// Mitsubishi GX Works2 project: R1R2 PLC Panel 20-08-2023_fr   PLC: Q03UDV

PROGRAM MAIN
; DEVICE NET
; OUTPUT LOGIC
; R1 TO R2 ZONE WAIT CLER
; R2 TO R1 ZONE
; CYCLE ON LOGIC
47    END
END_PROGRAM

PROGRAM CAMERA
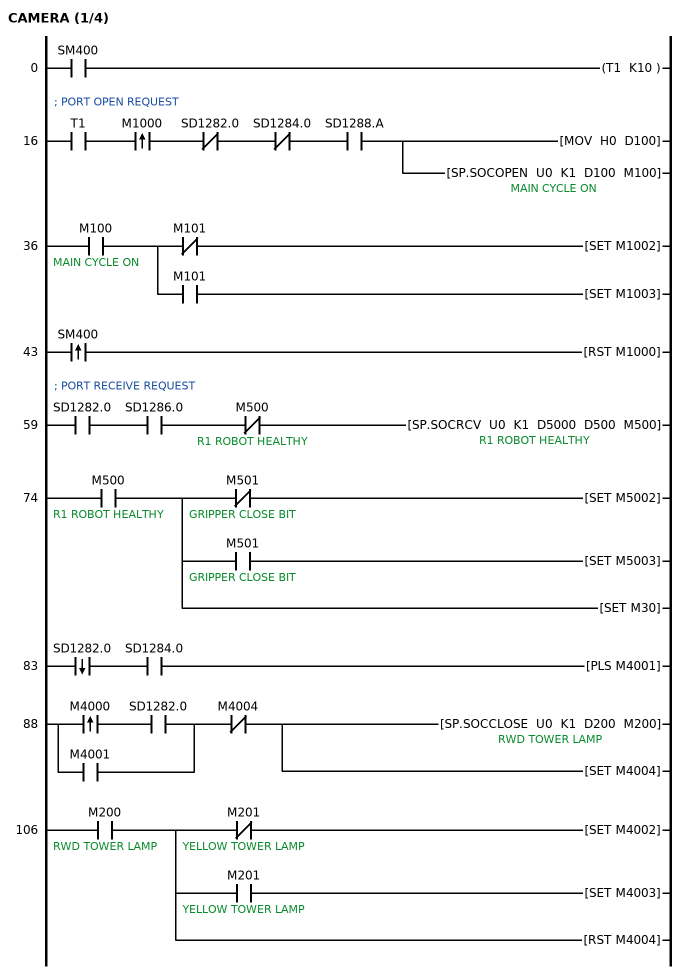
0     LD      SM400
      OUT     T1 K10
; PORT OPEN REQUEST
16    LD      T1
      ANDP    M1000
      ANI     SD1282.0
      ANI     SD1284.0
      AND     SD1288.A
      MOV     H0 D100
      SP.SOCOPEN U0 K1 D100 M100  ; MAIN CYCLE ON
36    LD      M100  ; MAIN CYCLE ON
      MPS
      ANI     M101
      SET     M1002
      MPP
      AND     M101
      SET     M1003
43    LDP     SM400
      RST     M1000
; PORT RECEIVE REQUEST
59    LD      SD1282.0
      AND     SD1286.0
      ANI     M500  ; R1 ROBOT HEALTHY
      SP.SOCRCV U0 K1 D5000 D500 M500
74    LD      M500  ; R1 ROBOT HEALTHY
      MPS
      ANI     M501  ; GRIPPER CLOSE BIT
      SET     M5002
      MRD
      AND     M501  ; GRIPPER CLOSE BIT
      SET     M5003
      MPP
      SET     M30
83    LDF     SD1282.0
      AND     SD1284.0
      PLS     M4001
88    LDP     M4000
      AND     SD1282.0
      OR      M4001
      ANI     M4004
      SP.SOCCLOSE U0 K1 D200 M200  ; RWD TOWER LAMP
      SET     M4004
106   LD      M200  ; RWD TOWER LAMP
      MPS
      ANI     M201  ; YELLOW TOWER LAMP
      SET     M4002
      MRD
      AND     M201  ; YELLOW TOWER LAMP
      SET     M4003
      MPP
      RST     M4004
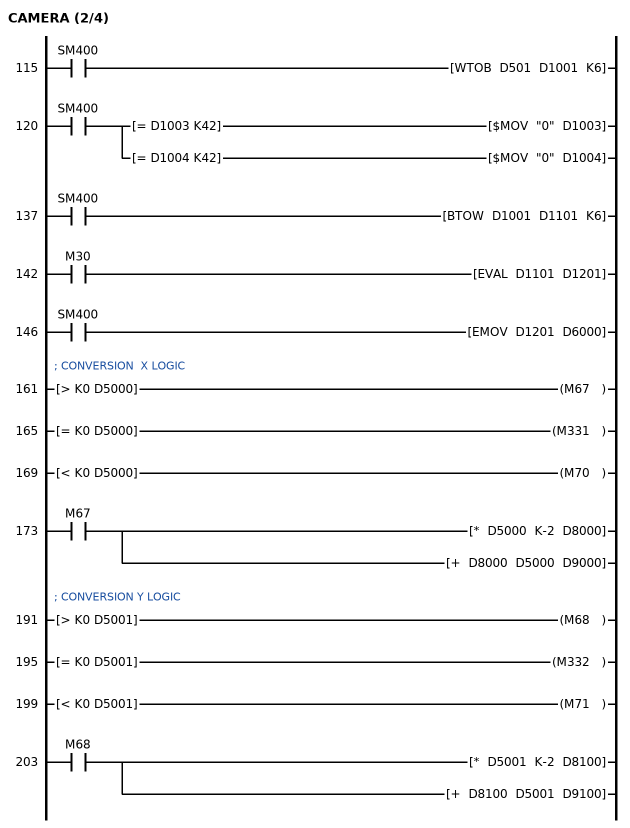
115   LD      SM400
      WTOB    D501 D1001 K6
120   LD      SM400
      MPS
      AND=    D1003 K42
      $MOV    "0" D1003
      MPP
      AND=    D1004 K42
      $MOV    "0" D1004
137   LD      SM400
      BTOW    D1001 D1101 K6
142   LD      M30
      EVAL    D1101 D1201
146   LD      SM400
      EMOV    D1201 D6000
; CONVERSION  X LOGIC
161   LD>     K0 D5000
      OUT     M67
165   LD=     K0 D5000
      OUT     M331
169   LD<     K0 D5000
      OUT     M70
173   LD      M67
      *       D5000 K-2 D8000
      +       D8000 D5000 D9000
; CONVERSION Y LOGIC
191   LD>     K0 D5001
      OUT     M68
195   LD=     K0 D5001
      OUT     M332
199   LD<     K0 D5001
      OUT     M71
203   LD      M68
      *       D5001 K-2 D8100
      +       D8100 D5001 D9100
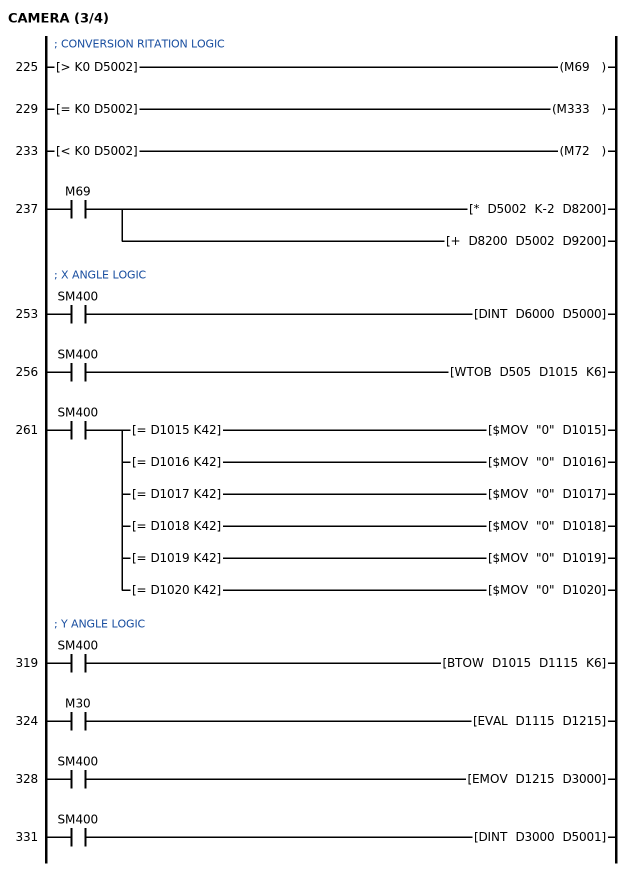
; CONVERSION RITATION LOGIC
225   LD>     K0 D5002
      OUT     M69
229   LD=     K0 D5002
      OUT     M333
233   LD<     K0 D5002
      OUT     M72
237   LD      M69
      *       D5002 K-2 D8200
      +       D8200 D5002 D9200
; X ANGLE LOGIC
253   LD      SM400
      DINT    D6000 D5000
256   LD      SM400
      WTOB    D505 D1015 K6
261   LD      SM400
      MPS
      AND=    D1015 K42
      $MOV    "0" D1015
      MRD
      AND=    D1016 K42
      $MOV    "0" D1016
      MRD
      AND=    D1017 K42
      $MOV    "0" D1017
      MRD
      AND=    D1018 K42
      $MOV    "0" D1018
      MRD
      AND=    D1019 K42
      $MOV    "0" D1019
      MPP
      AND=    D1020 K42
      $MOV    "0" D1020
; Y ANGLE LOGIC
319   LD      SM400
      BTOW    D1015 D1115 K6
324   LD      M30
      EVAL    D1115 D1215
328   LD      SM400
      EMOV    D1215 D3000
331   LD      SM400
      DINT    D3000 D5001
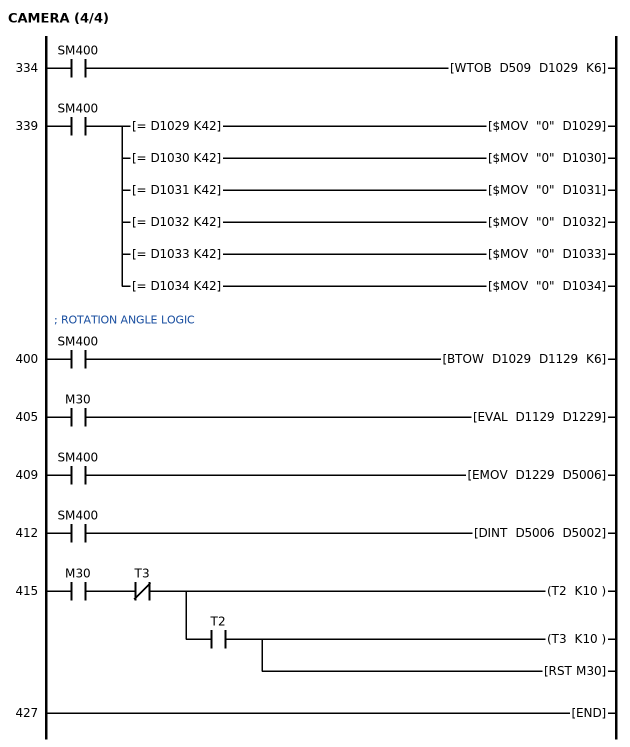
334   LD      SM400
      WTOB    D509 D1029 K6
339   LD      SM400
      MPS
      AND=    D1029 K42
      $MOV    "0" D1029
      MRD
      AND=    D1030 K42
      $MOV    "0" D1030
      MRD
      AND=    D1031 K42
      $MOV    "0" D1031
      MRD
      AND=    D1032 K42
      $MOV    "0" D1032
      MRD
      AND=    D1033 K42
      $MOV    "0" D1033
      MPP
      AND=    D1034 K42
      $MOV    "0" D1034
; ROTATION ANGLE LOGIC
400   LD      SM400
      BTOW    D1029 D1129 K6
405   LD      M30
      EVAL    D1129 D1229
409   LD      SM400
      EMOV    D1229 D5006
412   LD      SM400
      DINT    D5006 D5002
415   LD      M30
      ANI     T3
      OUT     T2 K10
      AND     T2
      OUT     T3 K10
      RST     M30
427   END
END_PROGRAM

PROGRAM AUTO
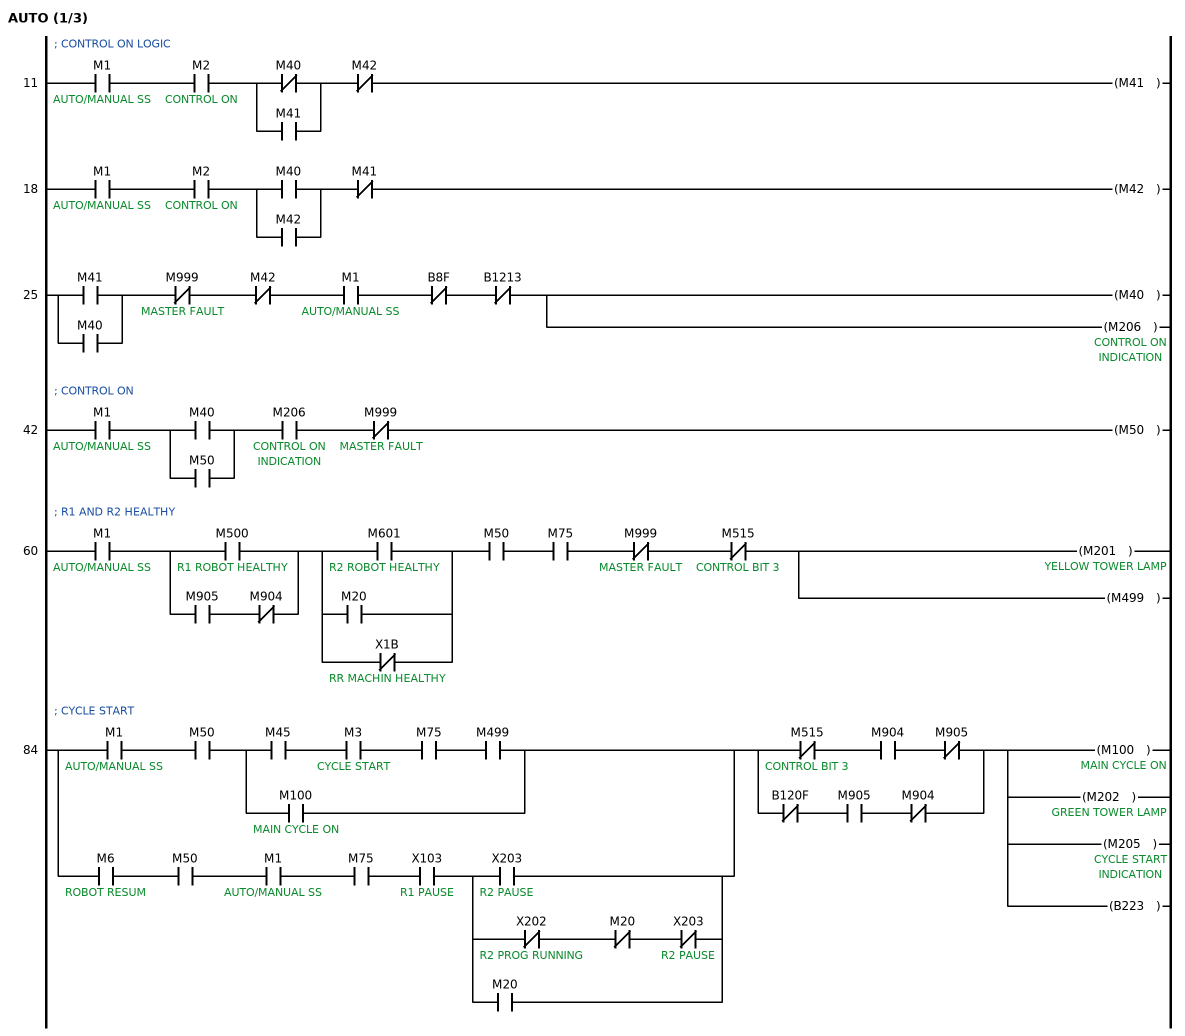
; CONTROL ON LOGIC
11    LD      M1  ; AUTO/MANUAL SS
      AND     M2  ; CONTROL ON
      LDI     M40
      OR      M41
      ANB
      ANI     M42
      OUT     M41
18    LD      M1  ; AUTO/MANUAL SS
      AND     M2  ; CONTROL ON
      LD      M40
      OR      M42
      ANB
      ANI     M41
      OUT     M42
25    LD      M41
      OR      M40
      ANI     M999  ; MASTER FAULT
      ANI     M42
      AND     M1  ; AUTO/MANUAL SS
      ANI     B8F
      ANI     B1213
      OUT     M40
      OUT     M206  ; CONTROL ON INDICATION
; CONTROL ON
42    LD      M1  ; AUTO/MANUAL SS
      LD      M40
      OR      M50
      ANB
      AND     M206  ; CONTROL ON INDICATION
      ANI     M999  ; MASTER FAULT
      OUT     M50
; R1 AND R2 HEALTHY
60    LD      M1  ; AUTO/MANUAL SS
      LD      M500  ; R1 ROBOT HEALTHY
      LD      M905
      ANI     M904
      ORB
      ANB
      LD      M601  ; R2 ROBOT HEALTHY
      OR      M20
      ORI     X1B  ; RR MACHIN HEALTHY
      ANB
      AND     M50
      AND     M75
      ANI     M999  ; MASTER FAULT
      ANI     M515  ; CONTROL BIT 3
      OUT     M201  ; YELLOW TOWER LAMP
      OUT     M499
; CYCLE START
84    LD      M1  ; AUTO/MANUAL SS
      AND     M50
      LD      M45
      AND     M3  ; CYCLE START
      AND     M75
      AND     M499
      OR      M100  ; MAIN CYCLE ON
      ANB
      LD      M6  ; ROBOT RESUM
      AND     M50
      AND     M1  ; AUTO/MANUAL SS
      AND     M75
      AND     X103  ; R1 PAUSE
      LD      X203  ; R2 PAUSE
      LDI     X202  ; R2 PROG RUNNING
      ANI     M20
      ANI     X203  ; R2 PAUSE
      ORB
      OR      M20
      ANB
      ORB
      LDI     M515  ; CONTROL BIT 3
      AND     M904
      ANI     M905
      LDI     B120F
      AND     M905
      ANI     M904
      ORB
      ANB
      OUT     M100  ; MAIN CYCLE ON
      OUT     M202  ; GREEN TOWER LAMP
      OUT     M205  ; CYCLE START INDICATION
      OUT     B223
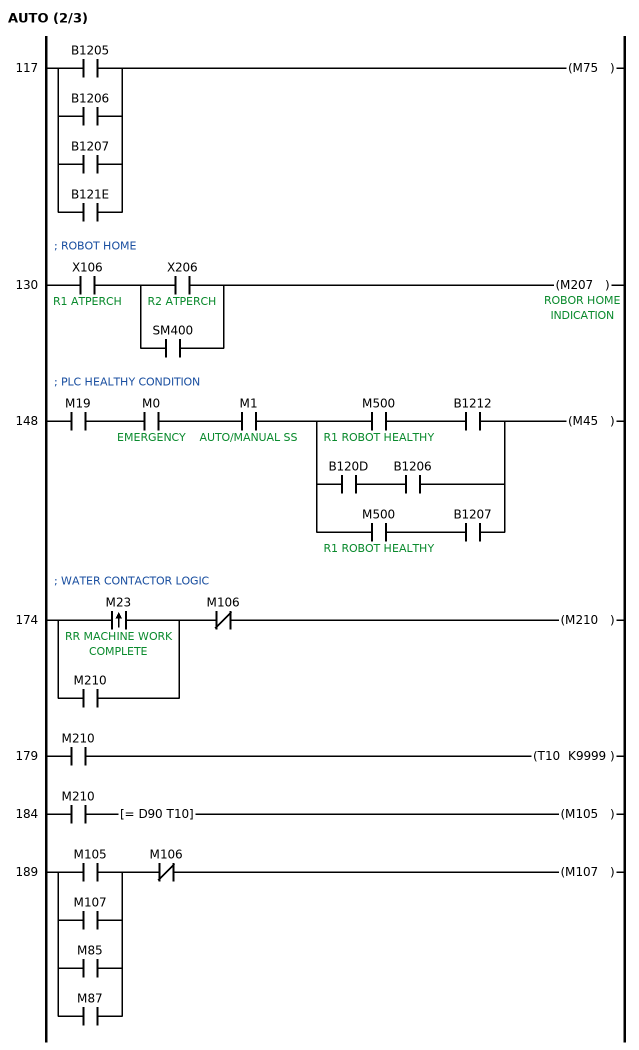
117   LD      B1205
      OR      B1206
      OR      B1207
      OR      B121E
      OUT     M75
; ROBOT HOME
130   LD      X106  ; R1 ATPERCH
      LD      X206  ; R2 ATPERCH
      OR      SM400
      ANB
      OUT     M207  ; ROBOR HOME INDICATION
; PLC HEALTHY CONDITION
148   LD      M19
      AND     M0  ; EMERGENCY
      AND     M1  ; AUTO/MANUAL SS
      LD      M500  ; R1 ROBOT HEALTHY
      AND     B1212
      LD      B120D
      AND     B1206
      ORB
      LD      M500  ; R1 ROBOT HEALTHY
      AND     B1207
      ORB
      ANB
      OUT     M45
; WATER CONTACTOR LOGIC
174   LDP     M23  ; RR MACHINE WORK COMPLETE
      OR      M210
      ANI     M106
      OUT     M210
179   LD      M210
      OUT     T10 K9999
184   LD      M210
      AND=    D90 T10
      OUT     M105
189   LD      M105
      OR      M107
      OR      M85
      OR      M87
      ANI     M106
      OUT     M107
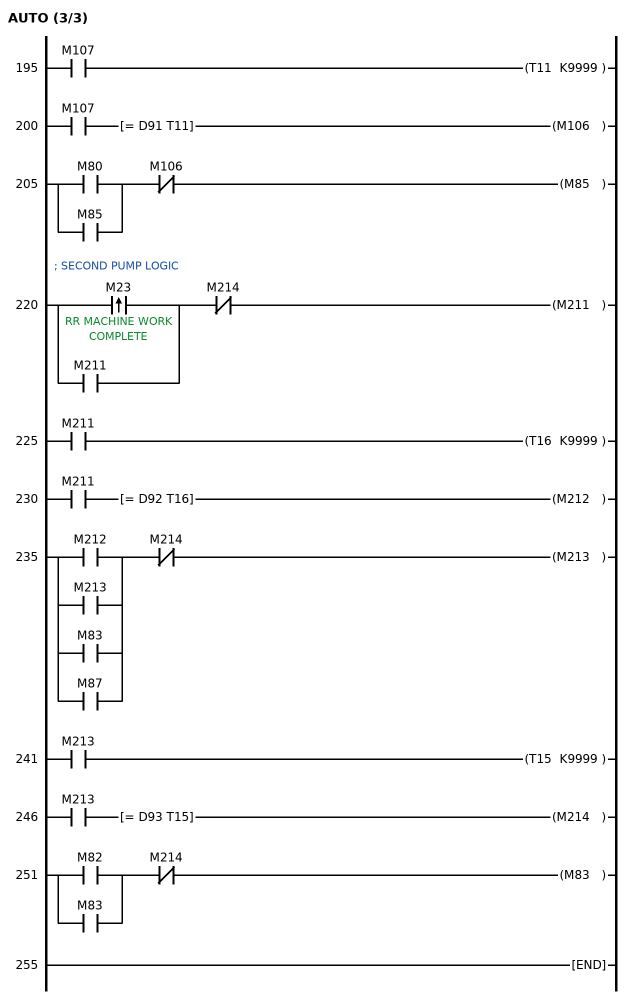
195   LD      M107
      OUT     T11 K9999
200   LD      M107
      AND=    D91 T11
      OUT     M106
205   LD      M80
      OR      M85
      ANI     M106
      OUT     M85
; SECOND PUMP LOGIC
220   LDP     M23  ; RR MACHINE WORK COMPLETE
      OR      M211
      ANI     M214
      OUT     M211
225   LD      M211
      OUT     T16 K9999
230   LD      M211
      AND=    D92 T16
      OUT     M212
235   LD      M212
      OR      M213
      OR      M83
      OR      M87
      ANI     M214
      OUT     M213
241   LD      M213
      OUT     T15 K9999
246   LD      M213
      AND=    D93 T15
      OUT     M214
251   LD      M82
      OR      M83
      ANI     M214
      OUT     M83
255   END
END_PROGRAM

PROGRAM CCLINK
0     END
END_PROGRAM

PROGRAM D-NET
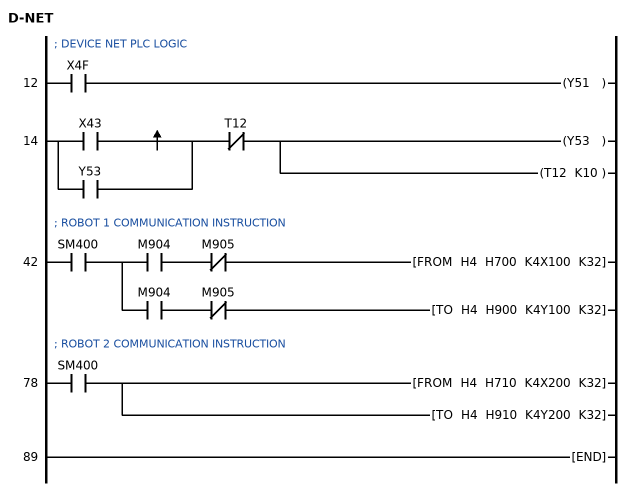
; DEVICE NET PLC LOGIC
12    LD      X4F
      OUT     Y51
14    LD      X43
      MEP
      OR      Y53
      ANI     T12
      OUT     Y53
      OUT     T12 K10
; ROBOT 1 COMMUNICATION INSTRUCTION
42    LD      SM400
      MPS
      AND     M904
      ANI     M905
      FROM    H4 H700 K4X100 K32  ; R1 CMD ENABLE
      MPP
      AND     M904
      ANI     M905
      TO      H4 H900 K4Y100 K32  ; R1 IMSTP
; ROBOT 2 COMMUNICATION INSTRUCTION
78    LD      SM400
      FROM    H4 H710 K4X200 K32  ; R2 CMD ENABLE
      TO      H4 H910 K4Y200 K32  ; R2 IMSTP
89    END
END_PROGRAM

PROGRAM FAULT
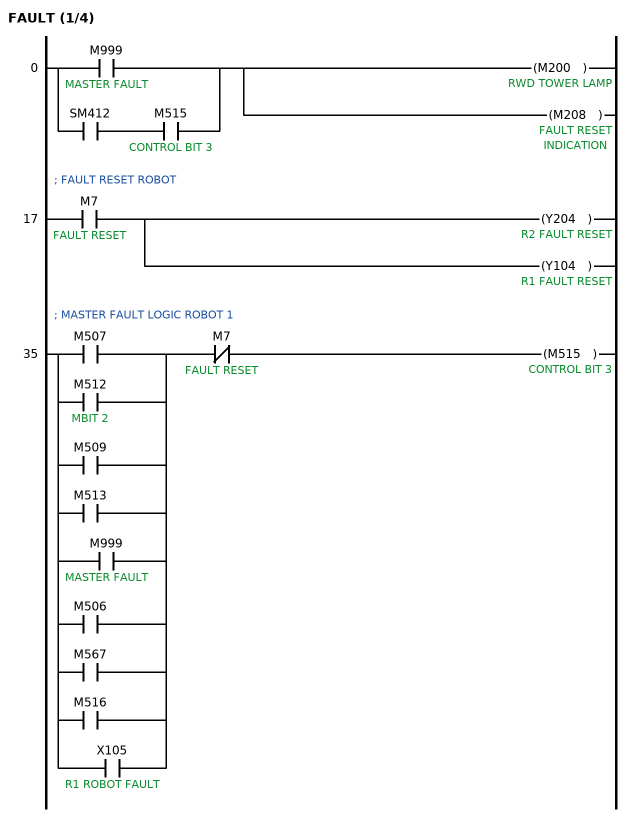
0     LD      M999  ; MASTER FAULT
      LD      SM412
      AND     M515  ; CONTROL BIT 3
      ORB
      OUT     M200  ; RWD TOWER LAMP
      OUT     M208  ; FAULT RESET INDICATION
; FAULT RESET ROBOT
17    LD      M7  ; FAULT RESET
      OUT     Y204  ; R2 FAULT RESET
      OUT     Y104  ; R1 FAULT RESET
; MASTER FAULT LOGIC ROBOT 1
35    LD      M507
      OR      M512  ; MBIT 2
      OR      M509
      OR      M513
      OR      M999  ; MASTER FAULT
      OR      M506
      OR      M567
      OR      M516
      OR      X105  ; R1 ROBOT FAULT
      ANI     M7  ; FAULT RESET
      OUT     M515  ; CONTROL BIT 3
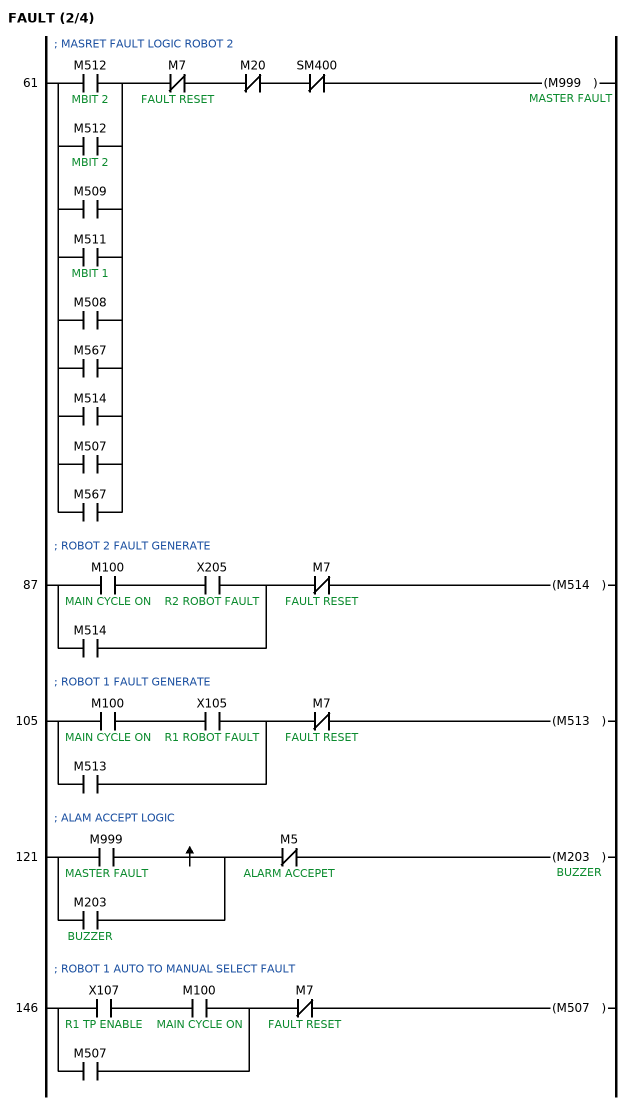
; MASRET FAULT LOGIC ROBOT 2
61    LD      M512  ; MBIT 2
      OR      M512  ; MBIT 2
      OR      M509
      OR      M511  ; MBIT 1
      OR      M508
      OR      M567
      OR      M514
      OR      M507
      OR      M567
      ANI     M7  ; FAULT RESET
      ANI     M20
      ANI     SM400
      OUT     M999  ; MASTER FAULT
; ROBOT 2 FAULT GENERATE
87    LD      M100  ; MAIN CYCLE ON
      AND     X205  ; R2 ROBOT FAULT
      OR      M514
      ANI     M7  ; FAULT RESET
      OUT     M514
; ROBOT 1 FAULT GENERATE
105   LD      M100  ; MAIN CYCLE ON
      AND     X105  ; R1 ROBOT FAULT
      OR      M513
      ANI     M7  ; FAULT RESET
      OUT     M513
; ALAM ACCEPT LOGIC
121   LD      M999  ; MASTER FAULT
      MEP
      OR      M203  ; BUZZER
      ANI     M5  ; ALARM ACCEPET
      OUT     M203  ; BUZZER
; ROBOT 1 AUTO TO MANUAL SELECT FAULT
146   LD      X107  ; R1 TP ENABLE
      AND     M100  ; MAIN CYCLE ON
      OR      M507
      ANI     M7  ; FAULT RESET
      OUT     M507
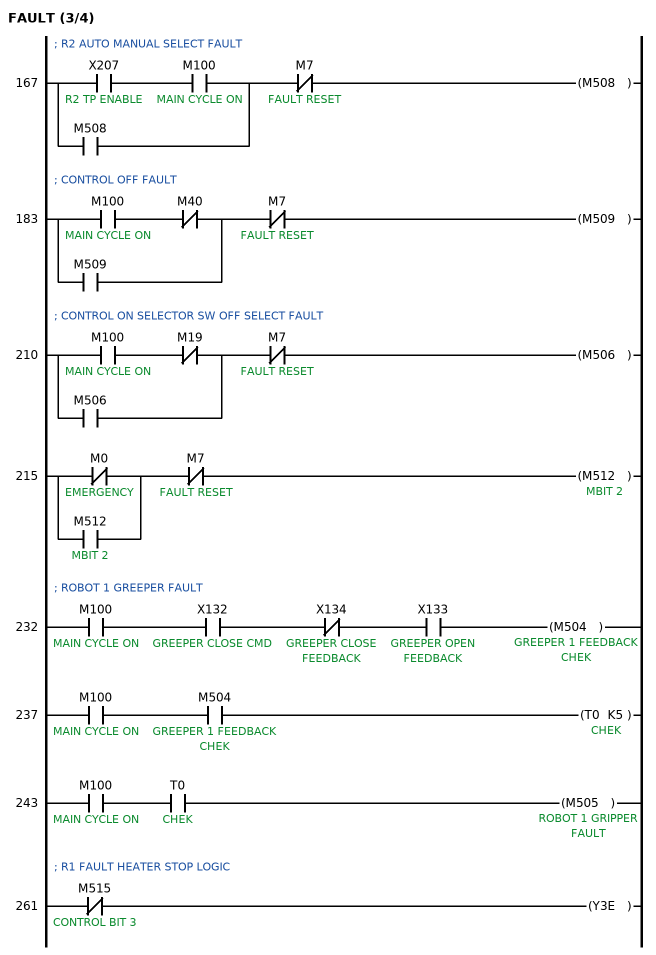
; R2 AUTO MANUAL SELECT FAULT
167   LD      X207  ; R2 TP ENABLE
      AND     M100  ; MAIN CYCLE ON
      OR      M508
      ANI     M7  ; FAULT RESET
      OUT     M508
; CONTROL OFF FAULT
183   LD      M100  ; MAIN CYCLE ON
      ANI     M40
      OR      M509
      ANI     M7  ; FAULT RESET
      OUT     M509
; CONTROL ON SELECTOR SW OFF SELECT FAULT
210   LD      M100  ; MAIN CYCLE ON
      ANI     M19
      OR      M506
      ANI     M7  ; FAULT RESET
      OUT     M506
215   LDI     M0  ; EMERGENCY
      OR      M512  ; MBIT 2
      ANI     M7  ; FAULT RESET
      OUT     M512  ; MBIT 2
; ROBOT 1 GREEPER FAULT
232   LD      M100  ; MAIN CYCLE ON
      AND     X132  ; GREEPER CLOSE CMD
      ANI     X134  ; GREEPER CLOSE FEEDBACK
      AND     X133  ; GREEPER OPEN FEEDBACK
      OUT     M504  ; GREEPER 1 FEEDBACK CHEK
237   LD      M100  ; MAIN CYCLE ON
      AND     M504  ; GREEPER 1 FEEDBACK CHEK
      OUT     T0 K5  ; CHEK
243   LD      M100  ; MAIN CYCLE ON
      AND     T0  ; CHEK
      OUT     M505  ; ROBOT 1 GRIPPER FAULT
; R1 FAULT HEATER STOP LOGIC
261   LDI     M515  ; CONTROL BIT 3
      OUT     Y3E
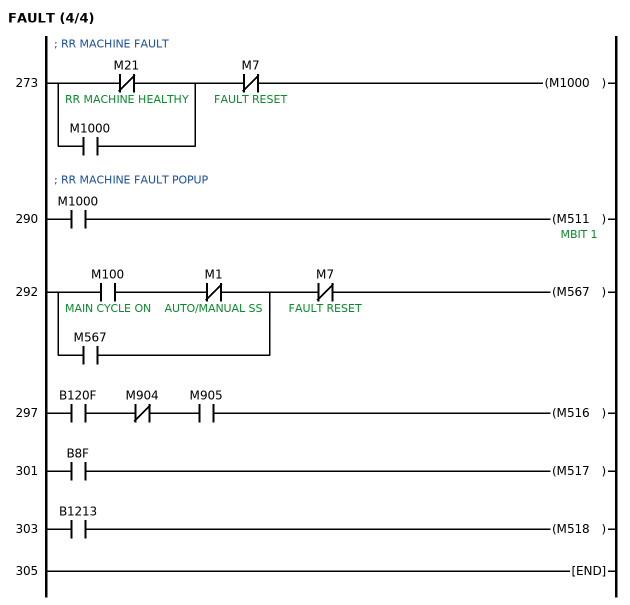
; RR MACHINE FAULT
273   LDI     M21  ; RR MACHINE HEALTHY
      OR      M1000
      ANI     M7  ; FAULT RESET
      OUT     M1000
; RR MACHINE FAULT POPUP
290   LD      M1000
      OUT     M511  ; MBIT 1
292   LD      M100  ; MAIN CYCLE ON
      ANI     M1  ; AUTO/MANUAL SS
      OR      M567
      ANI     M7  ; FAULT RESET
      OUT     M567
297   LD      B120F
      ANI     M904
      AND     M905
      OUT     M516
301   LD      B8F
      OUT     M517
303   LD      B1213
      OUT     M518
305   END
END_PROGRAM

PROGRAM INPUTMAP
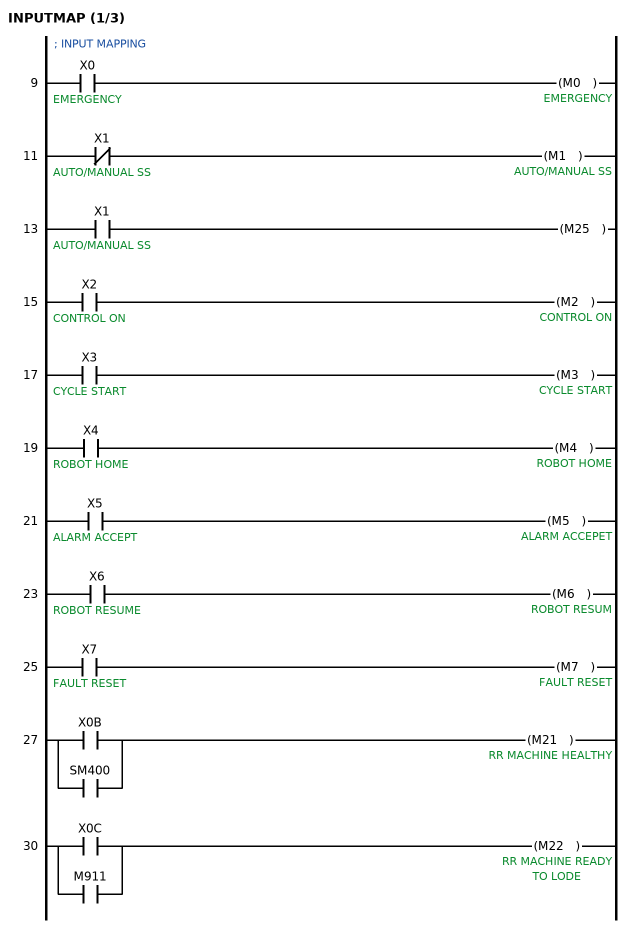
; INPUT MAPPING
9     LD      X0  ; EMERGENCY
      OUT     M0  ; EMERGENCY
11    LDI     X1  ; AUTO/MANUAL SS
      OUT     M1  ; AUTO/MANUAL SS
13    LD      X1  ; AUTO/MANUAL SS
      OUT     M25
15    LD      X2  ; CONTROL ON
      OUT     M2  ; CONTROL ON
17    LD      X3  ; CYCLE START
      OUT     M3  ; CYCLE START
19    LD      X4  ; ROBOT HOME
      OUT     M4  ; ROBOT HOME
21    LD      X5  ; ALARM ACCEPT
      OUT     M5  ; ALARM ACCEPET
23    LD      X6  ; ROBOT RESUME
      OUT     M6  ; ROBOT RESUM
25    LD      X7  ; FAULT RESET
      OUT     M7  ; FAULT RESET
27    LD      X0B
      OR      SM400
      OUT     M21  ; RR MACHINE HEALTHY
30    LD      X0C
      OR      M911
      OUT     M22  ; RR MACHINE READY TO LODE
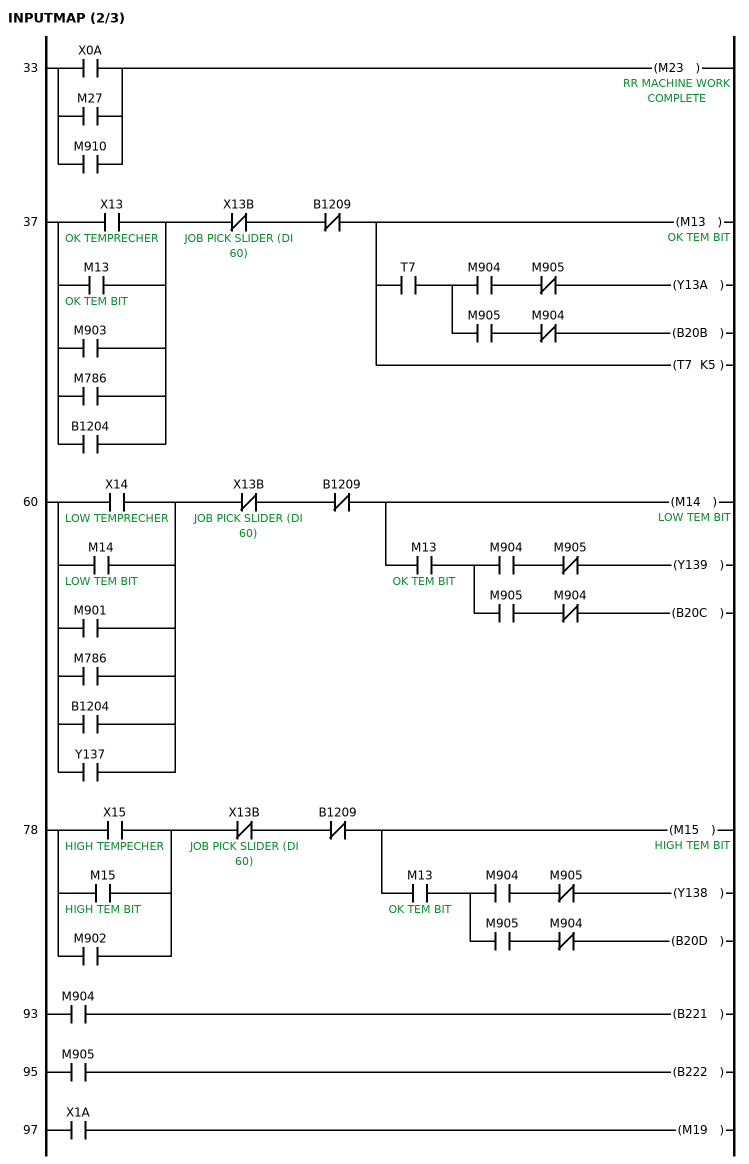
33    LD      X0A
      OR      M27
      OR      M910
      OUT     M23  ; RR MACHINE WORK COMPLETE
37    LD      X13  ; OK TEMPRECHER
      OR      M13  ; OK TEM BIT
      OR      M903
      OR      M786
      OR      B1204
      ANI     X13B  ; JOB PICK SLIDER (DI 60)
      ANI     B1209
      OUT     M13  ; OK TEM BIT
      MPS
      AND     T7
      MPS
      AND     M904
      ANI     M905
      OUT     Y13A
      MPP
      AND     M905
      ANI     M904
      OUT     B20B
      MPP
      OUT     T7 K5
60    LD      X14  ; LOW TEMPRECHER
      OR      M14  ; LOW TEM BIT
      OR      M901
      OR      M786
      OR      B1204
      OR      Y137
      ANI     X13B  ; JOB PICK SLIDER (DI 60)
      ANI     B1209
      OUT     M14  ; LOW TEM BIT
      AND     M13  ; OK TEM BIT
      MPS
      AND     M904
      ANI     M905
      OUT     Y139
      MPP
      AND     M905
      ANI     M904
      OUT     B20C
78    LD      X15  ; HIGH TEMPECHER
      OR      M15  ; HIGH TEM BIT
      OR      M902
      ANI     X13B  ; JOB PICK SLIDER (DI 60)
      ANI     B1209
      OUT     M15  ; HIGH TEM BIT
      AND     M13  ; OK TEM BIT
      MPS
      AND     M904
      ANI     M905
      OUT     Y138
      MPP
      AND     M905
      ANI     M904
      OUT     B20D
93    LD      M904
      OUT     B221
95    LD      M905
      OUT     B222
97    LD      X1A
      OUT     M19
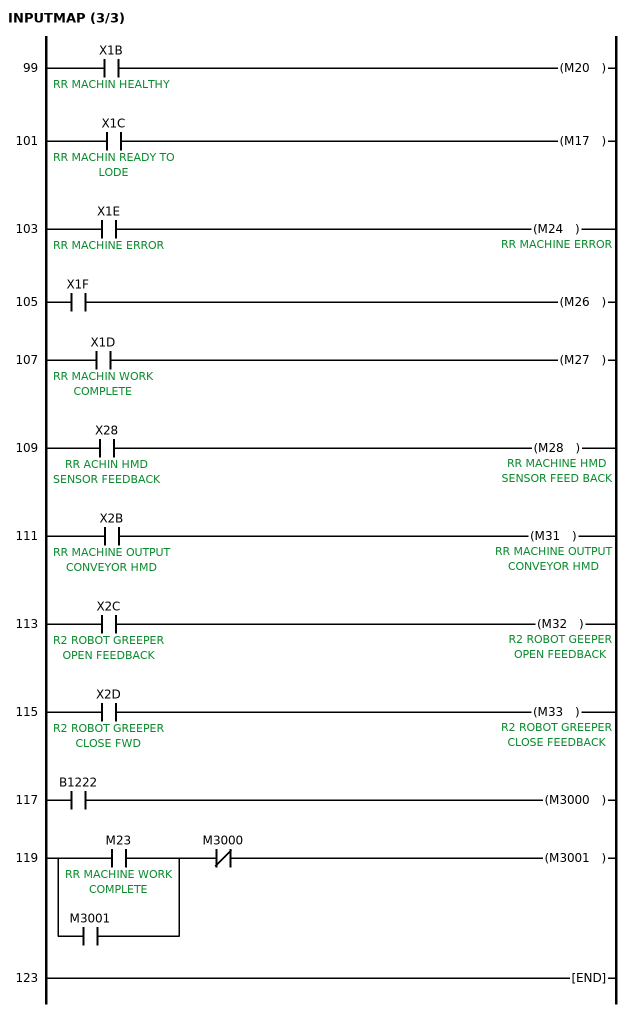
99    LD      X1B  ; RR MACHIN HEALTHY
      OUT     M20
101   LD      X1C  ; RR MACHIN READY TO LODE
      OUT     M17
103   LD      X1E  ; RR MACHINE ERROR
      OUT     M24  ; RR MACHINE ERROR
105   LD      X1F
      OUT     M26
107   LD      X1D  ; RR MACHIN WORK COMPLETE
      OUT     M27
109   LD      X28  ; RR ACHIN HMD SENSOR FEEDBACK
      OUT     M28  ; RR MACHINE HMD SENSOR FEED BACK
111   LD      X2B  ; RR MACHINE OUTPUT CONVEYOR HMD
      OUT     M31  ; RR MACHINE OUTPUT CONVEYOR HMD
113   LD      X2C  ; R2 ROBOT GREEPER OPEN FEEDBACK
      OUT     M32  ; R2 ROBOT GEEPER OPEN FEEDBACK
115   LD      X2D  ; R2 ROBOT GREEPER CLOSE FWD
      OUT     M33  ; R2 ROBOT GREEPER CLOSE FEEDBACK
117   LD      B1222
      OUT     M3000
119   LD      M23  ; RR MACHINE WORK COMPLETE
      OR      M3001
      ANI     M3000
      OUT     M3001
123   END
END_PROGRAM

PROGRAM MANUAL
0     END
END_PROGRAM

PROGRAM OUTPUTMA
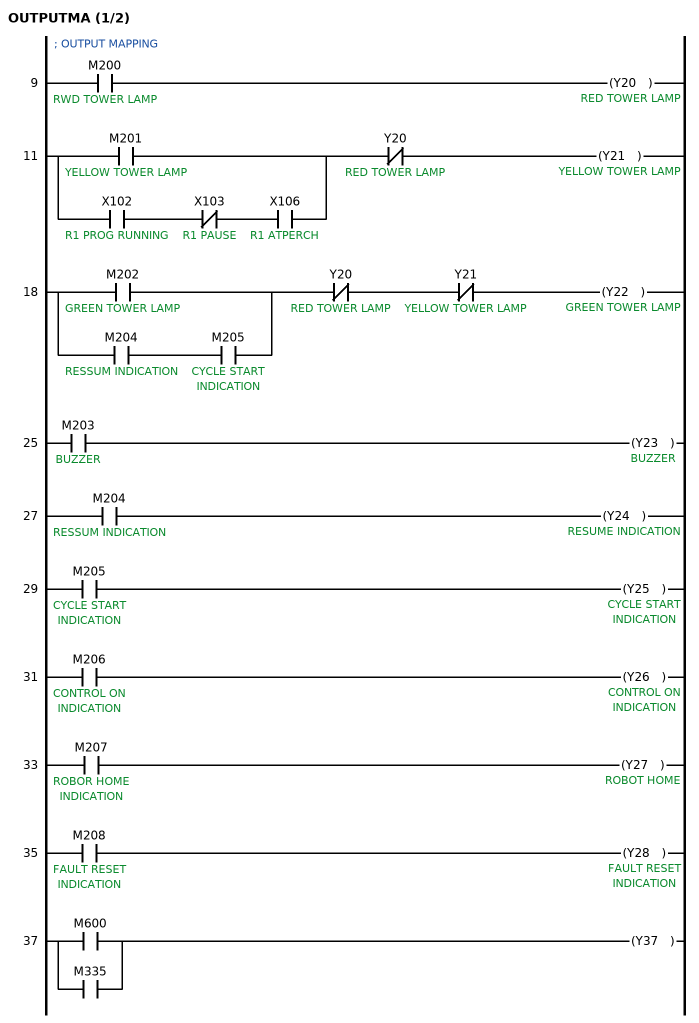
; OUTPUT MAPPING
9     LD      M200  ; RWD TOWER LAMP
      OUT     Y20  ; RED TOWER LAMP
11    LD      M201  ; YELLOW TOWER LAMP
      LD      X102  ; R1 PROG RUNNING
      ANI     X103  ; R1 PAUSE
      AND     X106  ; R1 ATPERCH
      ORB
      ANI     Y20  ; RED TOWER LAMP
      OUT     Y21  ; YELLOW TOWER LAMP
18    LD      M202  ; GREEN TOWER LAMP
      LD      M204  ; RESSUM INDICATION
      AND     M205  ; CYCLE START INDICATION
      ORB
      ANI     Y20  ; RED TOWER LAMP
      ANI     Y21  ; YELLOW TOWER LAMP
      OUT     Y22  ; GREEN TOWER LAMP
25    LD      M203  ; BUZZER
      OUT     Y23  ; BUZZER
27    LD      M204  ; RESSUM INDICATION
      OUT     Y24  ; RESUME INDICATION
29    LD      M205  ; CYCLE START INDICATION
      OUT     Y25  ; CYCLE START  INDICATION
31    LD      M206  ; CONTROL ON INDICATION
      OUT     Y26  ; CONTROL ON INDICATION
33    LD      M207  ; ROBOR HOME INDICATION
      OUT     Y27  ; ROBOT HOME
35    LD      M208  ; FAULT RESET INDICATION
      OUT     Y28  ; FAULT RESET INDICATION
37    LD      M600
      OR      M335
      OUT     Y37
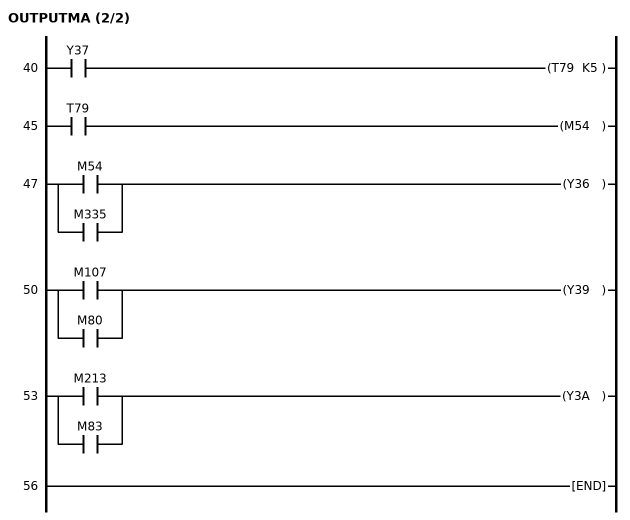
40    LD      Y37
      OUT     T79 K5
45    LD      T79
      OUT     M54
47    LD      M54
      OR      M335
      OUT     Y36
50    LD      M107
      OR      M80
      OUT     Y39
53    LD      M213
      OR      M83
      OUT     Y3A
56    END
END_PROGRAM

PROGRAM ROBO_1
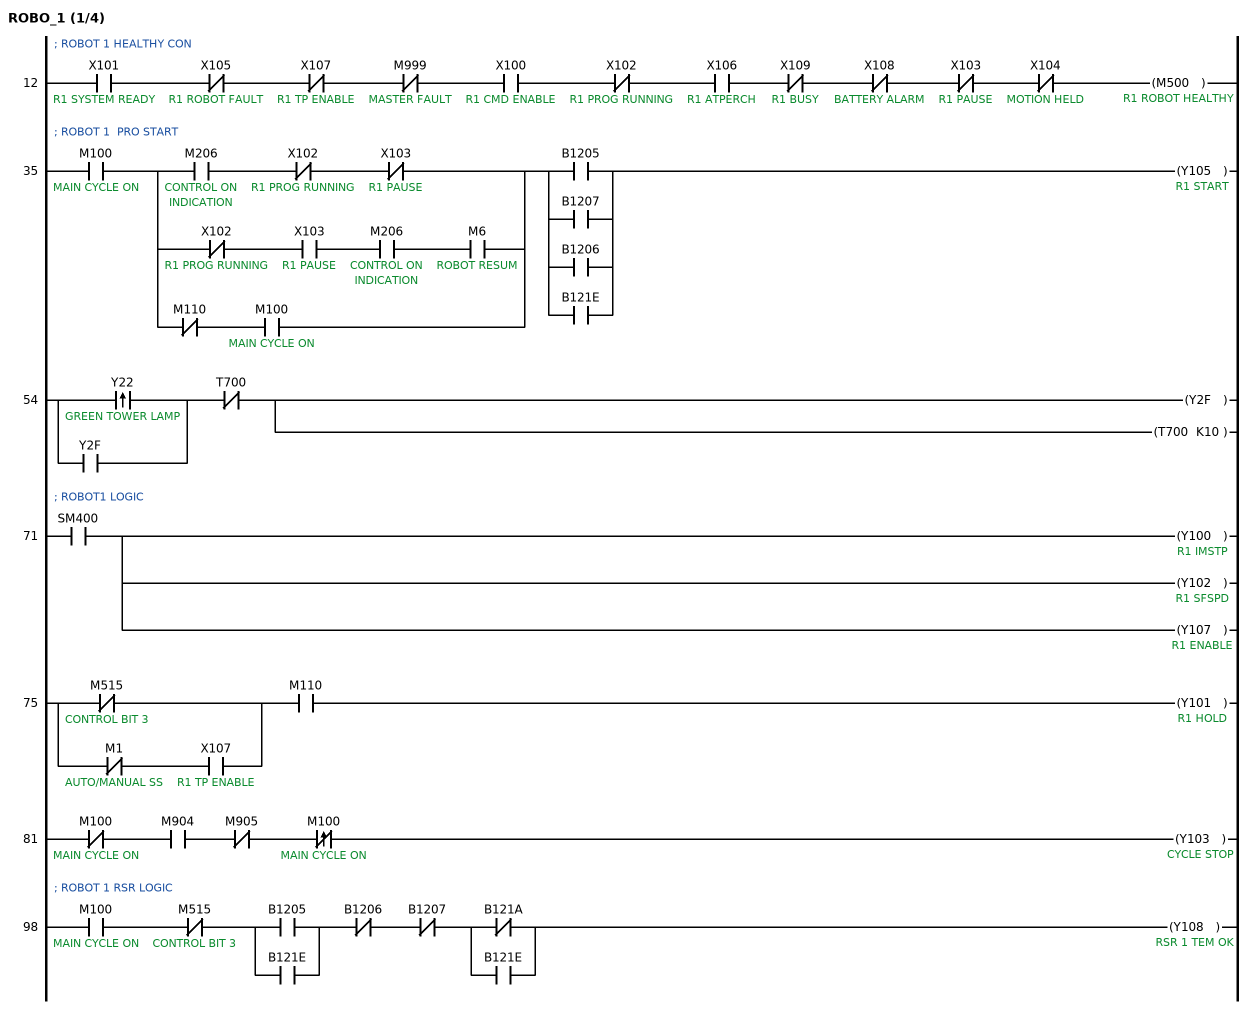
; ROBOT 1 HEALTHY CON
12    LD      X101  ; R1 SYSTEM READY
      ANI     X105  ; R1 ROBOT FAULT
      ANI     X107  ; R1 TP ENABLE
      ANI     M999  ; MASTER FAULT
      AND     X100  ; R1 CMD ENABLE
      ANI     X102  ; R1 PROG RUNNING
      AND     X106  ; R1 ATPERCH
      ANI     X109  ; R1 BUSY
      ANI     X108  ; BATTERY ALARM
      ANI     X103  ; R1 PAUSE
      ANI     X104  ; MOTION HELD
      OUT     M500  ; R1 ROBOT HEALTHY
; ROBOT 1  PRO START
35    LD      M100  ; MAIN CYCLE ON
      LD      M206  ; CONTROL ON INDICATION
      ANI     X102  ; R1 PROG RUNNING
      ANI     X103  ; R1 PAUSE
      LDI     X102  ; R1 PROG RUNNING
      AND     X103  ; R1 PAUSE
      AND     M206  ; CONTROL ON INDICATION
      AND     M6  ; ROBOT RESUM
      ORB
      LDI     M110
      AND     M100  ; MAIN CYCLE ON
      ORB
      ANB
      LD      B1205
      OR      B1207
      OR      B1206
      OR      B121E
      ANB
      OUT     Y105  ; R1 START
54    LDP     Y22  ; GREEN TOWER LAMP
      OR      Y2F
      ANI     T700
      OUT     Y2F
      OUT     T700 K10
; ROBOT1 LOGIC
71    LD      SM400
      OUT     Y100  ; R1 IMSTP
      OUT     Y102  ; R1 SFSPD
      OUT     Y107  ; R1 ENABLE
75    LDI     M515  ; CONTROL BIT 3
      LDI     M1  ; AUTO/MANUAL SS
      AND     X107  ; R1 TP ENABLE
      ORB
      AND     M110
      OUT     Y101  ; R1 HOLD
81    LDI     M100  ; MAIN CYCLE ON
      AND     M904
      ANI     M905
      ANDPI   M100  ; MAIN CYCLE ON
      OUT     Y103  ; CYCLE STOP
; ROBOT 1 RSR LOGIC
98    LD      M100  ; MAIN CYCLE ON
      ANI     M515  ; CONTROL BIT 3
      LD      B1205
      OR      B121E
      ANB
      ANI     B1206
      ANI     B1207
      LDI     B121A
      OR      B121E
      ANB
      OUT     Y108  ; RSR 1 TEM OK
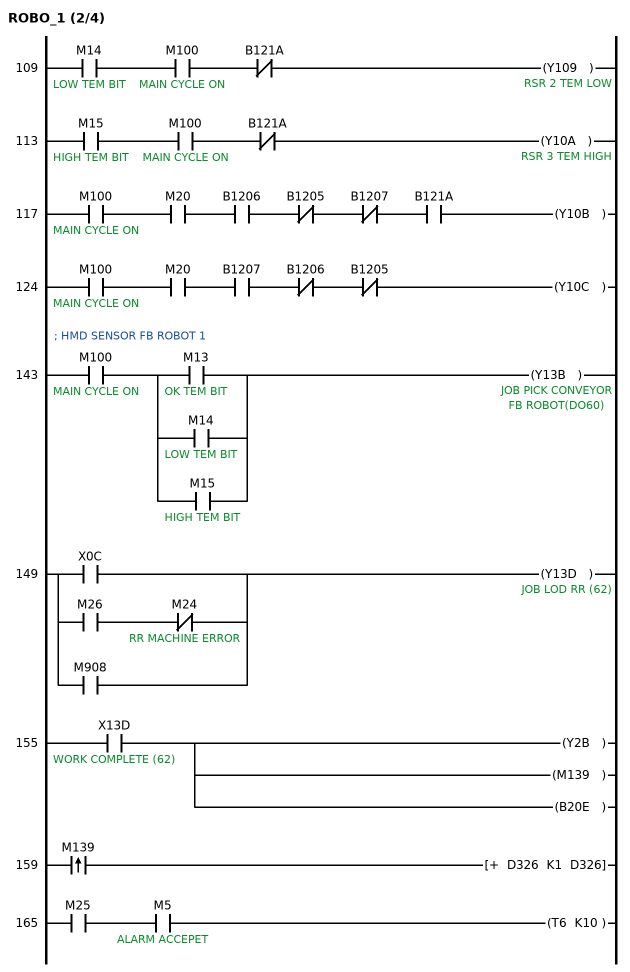
109   LD      M14  ; LOW TEM BIT
      AND     M100  ; MAIN CYCLE ON
      ANI     B121A
      OUT     Y109  ; RSR 2 TEM LOW
113   LD      M15  ; HIGH TEM BIT
      AND     M100  ; MAIN CYCLE ON
      ANI     B121A
      OUT     Y10A  ; RSR 3 TEM HIGH
117   LD      M100  ; MAIN CYCLE ON
      AND     M20
      AND     B1206
      ANI     B1205
      ANI     B1207
      AND     B121A
      OUT     Y10B
124   LD      M100  ; MAIN CYCLE ON
      AND     M20
      AND     B1207
      ANI     B1206
      ANI     B1205
      OUT     Y10C
; HMD SENSOR FB ROBOT 1
143   LD      M100  ; MAIN CYCLE ON
      LD      M13  ; OK TEM BIT
      OR      M14  ; LOW TEM BIT
      OR      M15  ; HIGH TEM BIT
      ANB
      OUT     Y13B  ; JOB PICK CONVEYOR FB ROBOT(DO60)
149   LD      X0C
      LD      M26
      ANI     M24  ; RR MACHINE ERROR
      ORB
      OR      M908
      OUT     Y13D  ; JOB LOD RR (62)
155   LD      X13D  ; WORK COMPLETE (62)
      OUT     Y2B
      OUT     M139
      OUT     B20E
159   LDP     M139
      +       D326 K1 D326
165   LD      M25
      AND     M5  ; ALARM ACCEPET
      OUT     T6 K10
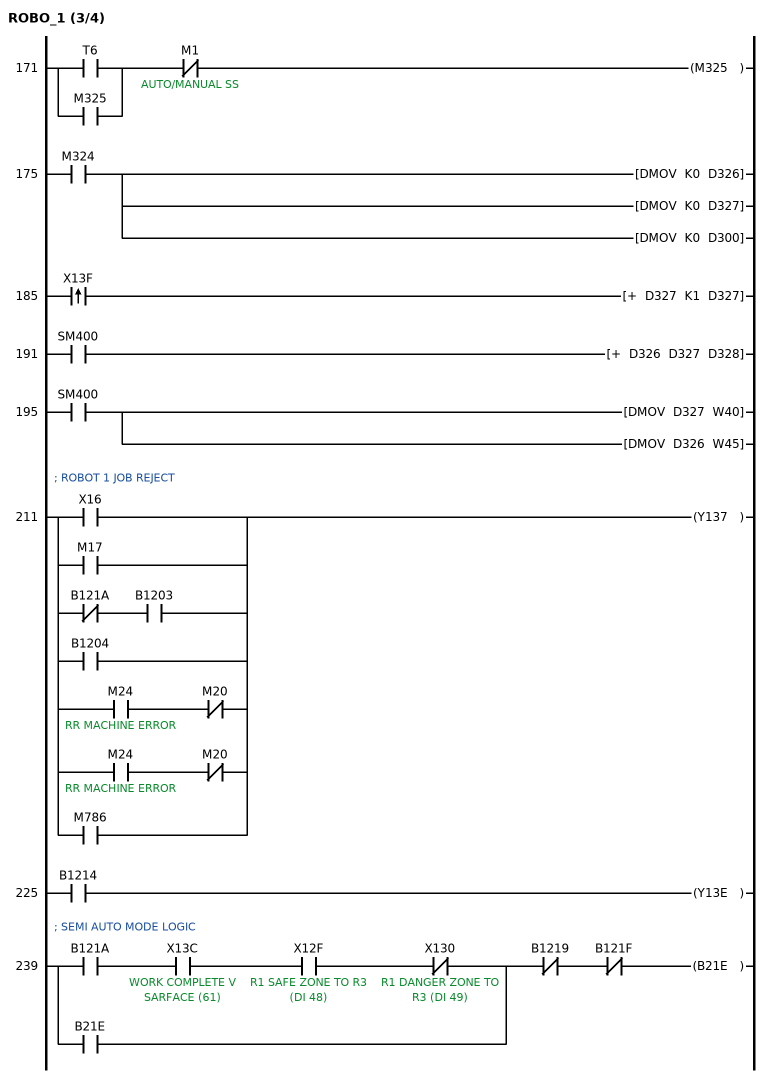
171   LD      T6
      OR      M325
      ANI     M1  ; AUTO/MANUAL SS
      OUT     M325
175   LD      M324
      DMOV    K0 D326
      DMOV    K0 D327
      DMOV    K0 D300
185   LDP     X13F
      +       D327 K1 D327
191   LD      SM400
      +       D326 D327 D328
195   LD      SM400
      DMOV    D327 W40
      DMOV    D326 W45
; ROBOT 1 JOB REJECT
211   LD      X16
      OR      M17
      LDI     B121A
      AND     B1203
      ORB
      OR      B1204
      LD      M24  ; RR MACHINE ERROR
      ANI     M20
      ORB
      LD      M24  ; RR MACHINE ERROR
      ANI     M20
      ORB
      OR      M786
      OUT     Y137
225   LD      B1214
      OUT     Y13E
; SEMI AUTO MODE LOGIC
239   LD      B121A
      AND     X13C  ; WORK COMPLETE V SARFACE (61)
      AND     X12F  ; R1 SAFE ZONE TO R3 (DI 48)
      ANI     X130  ; R1 DANGER ZONE TO R3 (DI 49)
      OR      B21E
      ANI     B1219
      ANI     B121F
      OUT     B21E
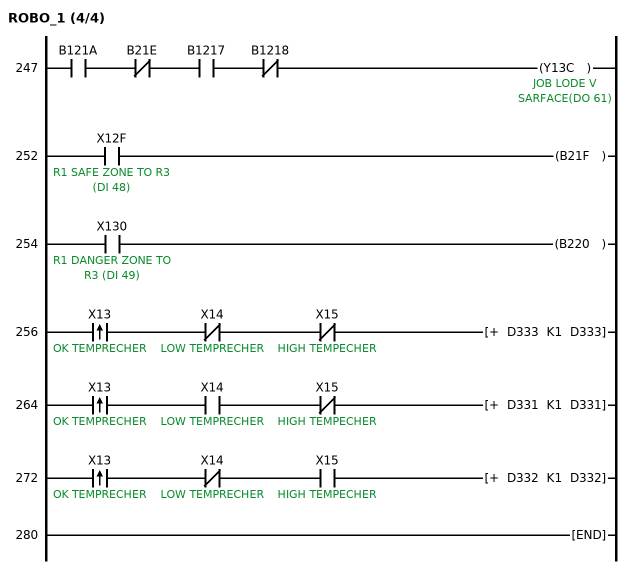
247   LD      B121A
      ANI     B21E
      AND     B1217
      ANI     B1218
      OUT     Y13C  ; JOB LODE V SARFACE(DO 61)
252   LD      X12F  ; R1 SAFE ZONE TO R3 (DI 48)
      OUT     B21F
254   LD      X130  ; R1 DANGER ZONE TO R3 (DI 49)
      OUT     B220
256   LDP     X13  ; OK TEMPRECHER
      ANI     X14  ; LOW TEMPRECHER
      ANI     X15  ; HIGH TEMPECHER
      +       D333 K1 D333
264   LDP     X13  ; OK TEMPRECHER
      AND     X14  ; LOW TEMPRECHER
      ANI     X15  ; HIGH TEMPECHER
      +       D331 K1 D331
272   LDP     X13  ; OK TEMPRECHER
      ANI     X14  ; LOW TEMPRECHER
      AND     X15  ; HIGH TEMPECHER
      +       D332 K1 D332
280   END
END_PROGRAM

PROGRAM ROBO_2
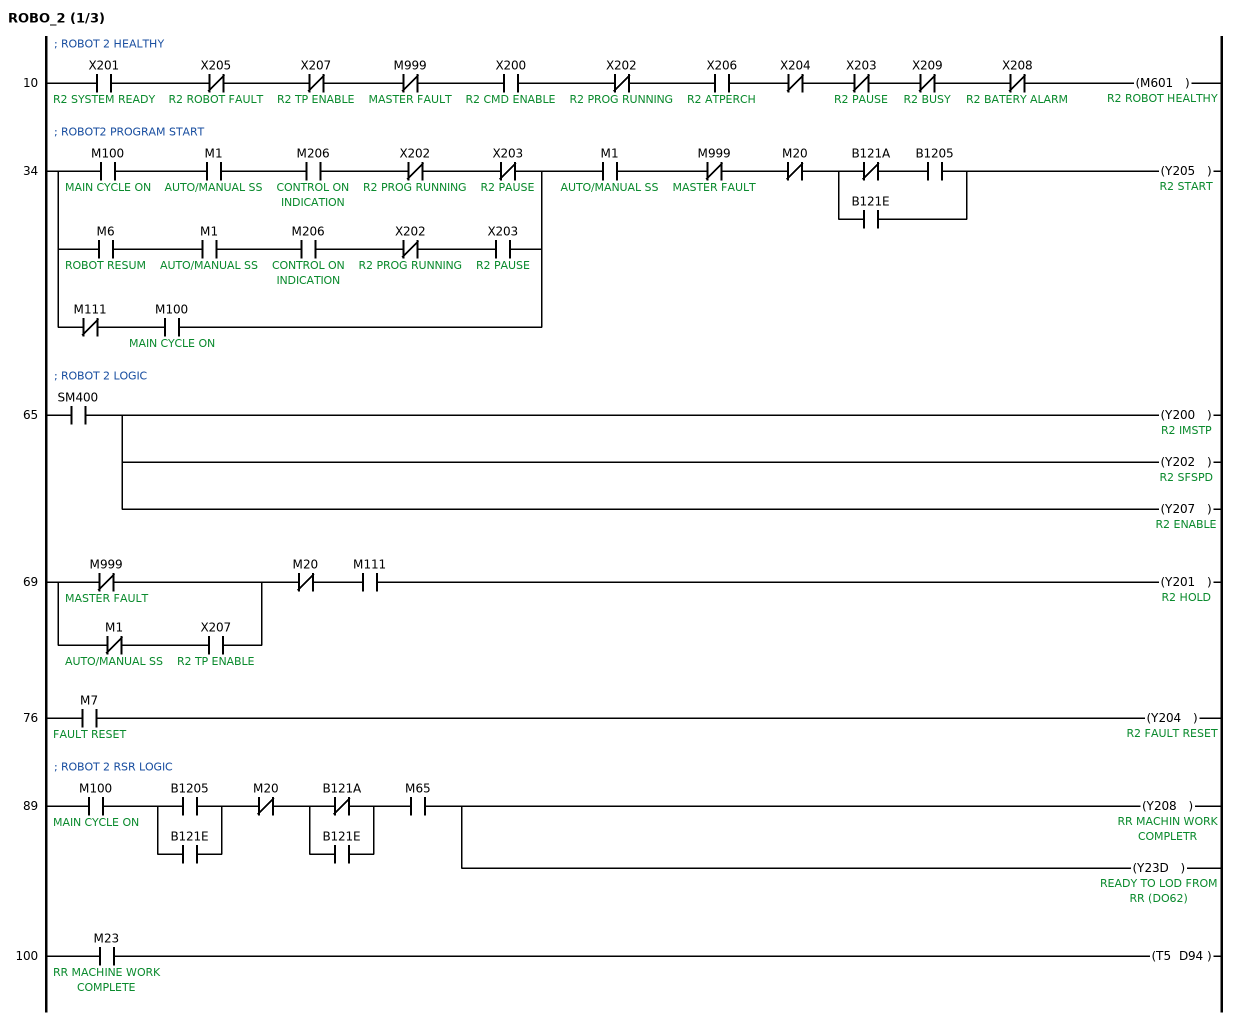
; ROBOT 2 HEALTHY
10    LD      X201  ; R2 SYSTEM READY
      ANI     X205  ; R2 ROBOT FAULT
      ANI     X207  ; R2 TP ENABLE
      ANI     M999  ; MASTER FAULT
      AND     X200  ; R2 CMD ENABLE
      ANI     X202  ; R2 PROG RUNNING
      AND     X206  ; R2 ATPERCH
      ANI     X204
      ANI     X203  ; R2 PAUSE
      ANI     X209  ; R2 BUSY
      ANI     X208  ; R2 BATERY ALARM
      OUT     M601  ; R2 ROBOT HEALTHY
; ROBOT2 PROGRAM START
34    LD      M100  ; MAIN CYCLE ON
      AND     M1  ; AUTO/MANUAL SS
      AND     M206  ; CONTROL ON INDICATION
      ANI     X202  ; R2 PROG RUNNING
      ANI     X203  ; R2 PAUSE
      LD      M6  ; ROBOT RESUM
      AND     M1  ; AUTO/MANUAL SS
      AND     M206  ; CONTROL ON INDICATION
      ANI     X202  ; R2 PROG RUNNING
      AND     X203  ; R2 PAUSE
      ORB
      LDI     M111
      AND     M100  ; MAIN CYCLE ON
      ORB
      AND     M1  ; AUTO/MANUAL SS
      ANI     M999  ; MASTER FAULT
      ANI     M20
      LDI     B121A
      AND     B1205
      OR      B121E
      ANB
      OUT     Y205  ; R2 START
; ROBOT 2 LOGIC
65    LD      SM400
      OUT     Y200  ; R2 IMSTP
      OUT     Y202  ; R2 SFSPD
      OUT     Y207  ; R2 ENABLE
69    LDI     M999  ; MASTER FAULT
      LDI     M1  ; AUTO/MANUAL SS
      AND     X207  ; R2 TP ENABLE
      ORB
      ANI     M20
      AND     M111
      OUT     Y201  ; R2 HOLD
76    LD      M7  ; FAULT RESET
      OUT     Y204  ; R2 FAULT RESET
; ROBOT 2 RSR LOGIC
89    LD      M100  ; MAIN CYCLE ON
      LD      B1205
      OR      B121E
      ANB
      ANI     M20
      LDI     B121A
      OR      B121E
      ANB
      AND     M65
      OUT     Y208  ; RR MACHIN WORK COMPLETR
      OUT     Y23D  ; READY TO LOD FROM RR (DO62)
100   LD      M23  ; RR MACHINE WORK COMPLETE
      OUT     T5 D94
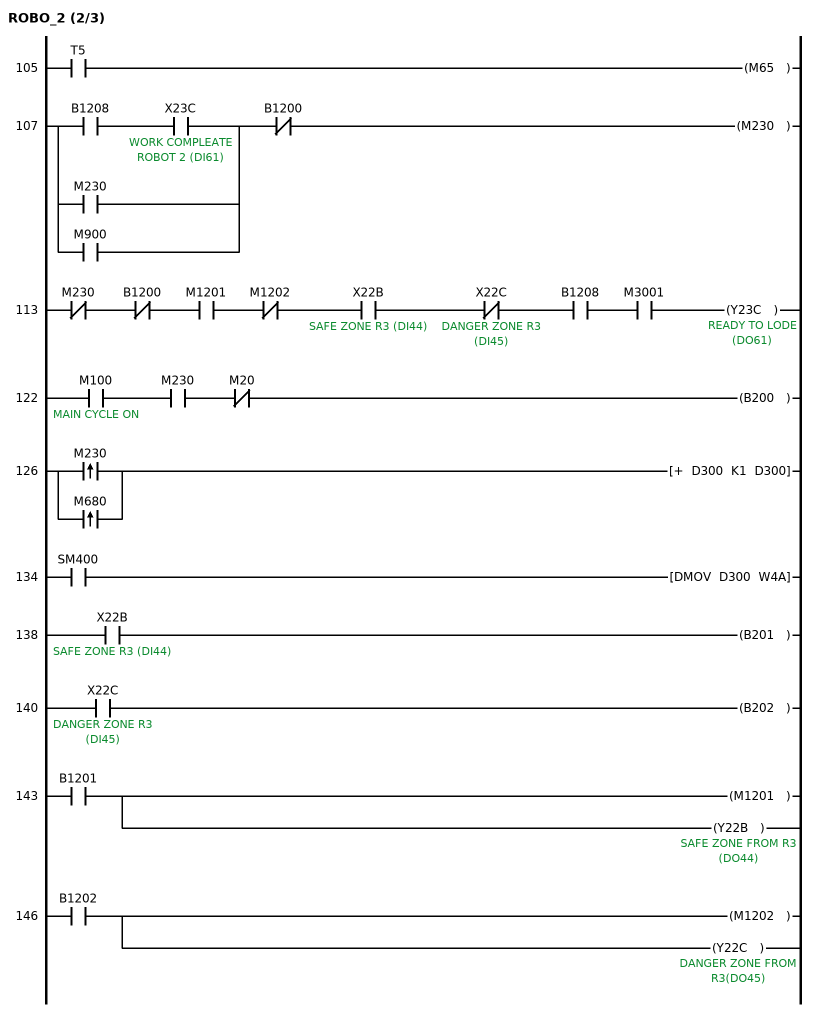
105   LD      T5
      OUT     M65
107   LD      B1208
      AND     X23C  ; WORK COMPLEATE ROBOT 2 (DI61)
      OR      M230
      OR      M900
      ANI     B1200
      OUT     M230
113   LDI     M230
      ANI     B1200
      AND     M1201
      ANI     M1202
      AND     X22B  ; SAFE ZONE R3 (DI44)
      ANI     X22C  ; DANGER ZONE R3 (DI45)
      AND     B1208
      AND     M3001
      OUT     Y23C  ; READY TO LODE  (DO61)
122   LD      M100  ; MAIN CYCLE ON
      AND     M230
      ANI     M20
      OUT     B200
126   LDP     M230
      ORP     M680
      +       D300 K1 D300
134   LD      SM400
      DMOV    D300 W4A
; 
138   LD      X22B  ; SAFE ZONE R3 (DI44)
      OUT     B201
140   LD      X22C  ; DANGER ZONE R3 (DI45)
      OUT     B202
; 
143   LD      B1201
      OUT     M1201
      OUT     Y22B  ; SAFE ZONE FROM R3 (DO44)
146   LD      B1202
      OUT     M1202
      OUT     Y22C  ; DANGER ZONE FROM R3(DO45)
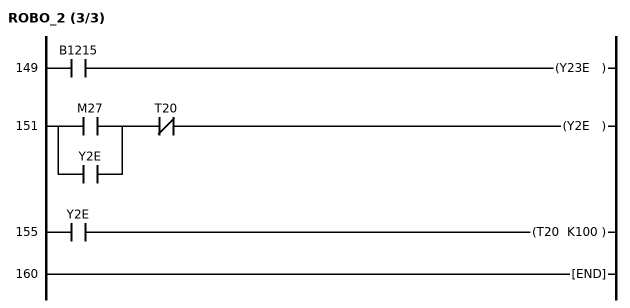
149   LD      B1215
      OUT     Y23E
151   LD      M27
      OR      Y2E
      ANI     T20
      OUT     Y2E
155   LD      Y2E
      OUT     T20 K100
160   END
END_PROGRAM

PROGRAM CC_LINK
